Fanuc TP program (LS listing): Animation_Pick.ls

/PROG  Animation_Pick
/ATTR
OWNER       = MNEDITOR;
COMMENT     = ""
PROG_SIZE   = 913;
CREATE      = DATE 25-11-29  TIME 15:54:19;
MODIFIED      = DATE 25-11-29  TIME 15:54:19;
FILE_NAME   = ;
VERSION    = 0;
LINE_COUNT  = 13;
MEMORY_SIZE = 1197;
PROTECT     = READ_WRITE;
TCD:  STACK_SIZE    = 0,
      TASK_PRIORITY = 50,
      TIME_SLICE    = 0,
      BUSY_LAMP_OFF = 0,
      ABORT_REQUEST = 0,
      PAUSE_REQUEST = 0;
DEFAULT_GROUP   = 1,*,*,*,*,*,*,* ;
CONTROL_CODE    = 00000000 00000000;
/APPL
AUTO_SINGULARITY_HEADER;
  ENABLE_SINGULARITY_AVOIDANCE	: TRUE;

/MN
1:!FANUC America Corp. ;
2:!ROBOGUIDE Generated This TPP ;
3:!Run SimPRO.cf to setup frame and tool data ;
4:!This program will be overwritten on the next save or run. ;
5:! Pickup ('cylinder') From ('re-grip_stand_HighQuality_Pick') With ('GP: 1 - UT: 1  (Hand)') ;
7:!WAIT 0.00 (sec) ;
/POS
/END
